Fanuc KAREL source: kc00007.KL

-- PROVISIONAL review KL for V1013-1; original PC SHA256 bf06fcbfb5c945ec738c1dbbb8f3e3c7750a73a690fd5326279fee48796730a7
-- Incomplete behavior may be omitted. Consult companion uncertainty JSON. Do not deploy.
PROGRAM KC00007
%NOLOCKGROUP
BEGIN
  -- UNRESOLVED_PC offsets 5-51; opcodes 27,22,1C,22,22,22,1C,22,31
  -- UNRESOLVED_PC offsets 56-60; opcodes 7F
END KC00007
